// TwinCAT 3 PLC project Plc
// ProgramVersion: 3.1.4024.0
// libraries:
//   Tc2_Standard, * (Beckhoff Automation GmbH)
//   Tc2_System, * (Beckhoff Automation GmbH)
//   Tc3_Module, * (Beckhoff Automation GmbH)
// project tree:
//   OOP/Elements/ I_PushButton.TcIO, I_Sensor.TcIO, NormallyOpenPushButton.TcPOU, NormallyClosePushButton.TcPOU, NormallyOpenSensor.TcPOU, NormallyCloseSensor.TcPOU
//   OOP/Module/ I_Motor.TcIO, MotorControl.TcPOU, SortingConveyor.TcPOU
//   OOP/ PRG_OOPApproach.TcPOU
//   / PlcTask.TcTTO
//   POUs/ MAIN.TcPOU, PRG_SortingConveyor_proceduralApproach.TcPOU

CONFIGURATION Plc
    RESOURCE PLC ON TwinCAT3
        TASK PlcTask(INTERVAL := T#10ms, PRIORITY := 20);
        PROGRAM MAIN WITH PlcTask : MAIN;
    END_RESOURCE
END_CONFIGURATION

// ---- OOP/Elements/I_PushButton.TcIO
INTERFACE I_PushButton

PROPERTY PUBLIC isPressed : BOOL
GET
END_GET
END_PROPERTY

PROPERTY PUBLIC isReleased : BOOL
GET
END_GET
END_PROPERTY

END_INTERFACE

// ---- OOP/Elements/I_Sensor.TcIO
INTERFACE I_Sensor

PROPERTY PUBLIC isActive : BOOL
GET
END_GET
END_PROPERTY

PROPERTY PUBLIC isInactive : BOOL
GET
END_GET
END_PROPERTY

END_INTERFACE

// ---- OOP/Module/I_Motor.TcIO
INTERFACE I_Motor

METHOD PUBLIC Start
VAR_INPUT
END_VAR
END_METHOD

METHOD PUBLIC stop : BOOL
VAR_INPUT
END_VAR
END_METHOD

END_INTERFACE

// ---- POUs/MAIN.TcPOU
PROGRAM MAIN
VAR

END_VAR


	PRG_SortingConveyor_proceduralApproach();
	PRG_OOPApproach();

END_PROGRAM

// ---- POUs/PRG_SortingConveyor_proceduralApproach.TcPOU
PROGRAM PRG_SortingConveyor_proceduralApproach
VAR
	stop AT%I* : BOOL;
	emergency AT%I* : BOOL;
	start AT%I* : BOOL;
	productDetectedSensor AT%I* : BOOL;
	conveyorFullSensor AT%I* : BOOL;
	motorContactor AT%Q* : BOOL;
	conveyorControl: BOOL;

	timeout: TOF;	
END_VAR

	
IF (NOT stop) OR (NOT emergency) THEN
	conveyorControl	:=	FALSE;
ELSIF start AND (stop) AND (emergency) THEN
	conveyorControl	:=	TRUE;
END_IF
	
timeout(IN:= conveyorControl AND productDetectedSensor, PT:= T#5S, Q=> , ET=> );

motorContactor	:=	conveyorControl AND timeout.Q AND (NOT conveyorFullSensor);

END_PROGRAM

// ---- OOP/PRG_OOPApproach.TcPOU
PROGRAM PRG_OOPApproach
VAR
	stop : NormallyClosePushButton;
	emergency : NormallyClosePushButton;
	stopNO : NormallyOpenPushButton;
	emergencyNO : NormallyOpenPushButton;
	start : NormallyOpenPushButton;
	productDetectedSensor : NormallyOpenSensor;
	conveyorFullSensor : NormallyOpenSensor;
	motorContactor : MotorControl;
	
	SortingConveyor: SortingConveyor (stop, emergency, start, productDetectedSensor, conveyorFullSensor, motorContactor);
	
//	conveyorControl: BOOL;
//	timeout: TOF;	
	
	
	useSpareSensor: BOOL;
END_VAR

	
IF NOT useSpareSensor THEN
	SortingConveyor (	
		stop:= stop, 
		emergency:= emergency, 
		start:= start, 
		productDetectedSensor:= productDetectedSensor, 
		conveyorFullSensor:= conveyorFullSensor, 
		motorContactor:= motorContactor	);
ELSE
	SortingConveyor (	
		stop:= stopNO, 
		emergency:= emergencyNO, 
		start:= start, 
		productDetectedSensor:= productDetectedSensor, 
		conveyorFullSensor:= conveyorFullSensor, 
		motorContactor:= motorContactor	);	
END_IF


//	IF (stop.isPressed) OR (emergency.isPressed) THEN
//		conveyorControl	:=	FALSE;
//	ELSIF start.isPressed AND (stop.isReleased) AND (emergency.isReleased) THEN
//		conveyorControl	:=	TRUE;
//	END_IF
		
//	timeout(IN:= conveyorControl AND productDetectedSensor.isActive, PT:= T#5S, Q=> , ET=> );

//	IF conveyorControl AND timeout.Q AND (conveyorFullSensor.isInactive) THEN
//		motorContactor.Start();	
//	ELSE
//		motorContactor.Stop();	
//	END_IF

END_PROGRAM

// ---- OOP/Elements/NormallyClosePushButton.TcPOU
FUNCTION_BLOCK NormallyClosePushButton IMPLEMENTS I_PushButton
VAR
	input AT%I* : BOOL;
END_VAR

PROPERTY PUBLIC isPressed : BOOL
GET
isPressed	:=	NOT input;
END_GET
END_PROPERTY

PROPERTY PUBLIC isReleased : BOOL
GET
isReleased	:=	input;
END_GET
END_PROPERTY

END_FUNCTION_BLOCK

// ---- OOP/Elements/NormallyOpenPushButton.TcPOU
FUNCTION_BLOCK NormallyOpenPushButton IMPLEMENTS I_PushButton
VAR
	input AT%I* : BOOL;
END_VAR

PROPERTY PUBLIC isPressed : BOOL
GET
isPressed	:=	input;
END_GET
END_PROPERTY

PROPERTY PUBLIC isReleased : BOOL
GET
isReleased	:=	NOT input;
END_GET
END_PROPERTY

END_FUNCTION_BLOCK

// ---- OOP/Elements/NormallyOpenSensor.TcPOU
FUNCTION_BLOCK NormallyOpenSensor IMPLEMENTS I_Sensor
VAR
	input AT%I* : BOOL;
END_VAR

PROPERTY PUBLIC isActive : BOOL
GET
isActive	:=	input;
END_GET
END_PROPERTY

PROPERTY PUBLIC isInactive : BOOL
GET
isInactive	:=	NOT input;
END_GET
END_PROPERTY

END_FUNCTION_BLOCK

// ---- OOP/Module/MotorControl.TcPOU
FUNCTION_BLOCK MotorControl IMPLEMENTS I_Motor
VAR
	OnOff AT%Q* : BOOL;
END_VAR

METHOD PUBLIC Start
VAR_INPUT
END_VAR
OnOff	:=	TRUE;
END_METHOD

METHOD PUBLIC stop : BOOL
VAR_INPUT
END_VAR
OnOff := FALSE;
END_METHOD

END_FUNCTION_BLOCK

// ---- OOP/Module/SortingConveyor.TcPOU
FUNCTION_BLOCK SortingConveyor
VAR_INPUT
	stop : I_PushButton;
	emergency : I_PushButton;
	start : I_PushButton;
	productDetectedSensor : I_Sensor;
	conveyorFullSensor : I_Sensor;
	motorContactor : I_Motor;
END_VAR
VAR_OUTPUT
END_VAR
VAR	
	conveyorControl: BOOL;
	timeout: TOF;		
	
END_VAR

		
	IF (stop.isPressed) OR (emergency.isPressed) THEN
		conveyorControl	:=	FALSE;
	ELSIF start.isPressed AND (stop.isReleased) AND (emergency.isReleased) THEN
		conveyorControl	:=	TRUE;
	END_IF
		
	timeout(IN:= conveyorControl AND productDetectedSensor.isActive, PT:= T#5S, Q=> , ET=> );

	IF conveyorControl AND timeout.Q AND (conveyorFullSensor.isInactive) THEN
		motorContactor.Start();	
	ELSE
		motorContactor.Stop();	
	END_IF

METHOD FB_init : BOOL
VAR_INPUT
	bInitRetains : BOOL; // if TRUE, the retain variables are initialized (warm start / cold start)
	bInCopyCode : BOOL;  // if TRUE, the instance afterwards gets moved into the copy code (online change)

	stop : I_PushButton;
	emergency : I_PushButton;
	start : I_PushButton;
	productDetectedSensor : I_Sensor;
	conveyorFullSensor : I_Sensor;
	motorContactor : I_Motor;
	
END_VAR

	THIS^.stop 						:=	stop 					; 
	THIS^.emergency 				:=  emergency 				;
	THIS^.start 					:=  start 					;
	THIS^.productDetectedSensor 	:=  productDetectedSensor 	;
	THIS^.conveyorFullSensor 		:=  conveyorFullSensor 		;
	THIS^.motorContactor 			:=  motorContactor 			;
END_METHOD

END_FUNCTION_BLOCK

// ---- OOP/Elements/NormallyCloseSensor.TcPOU
FUNCTION_BLOCK NormallyCloseSensor IMPLEMENTS I_Sensor
VAR
	input AT%I* : BOOL;
END_VAR

PROPERTY PUBLIC isActive : BOOL
GET
isActive	:=	NOT input;
END_GET
END_PROPERTY

PROPERTY PUBLIC isInactive : BOOL
GET
isInactive	:=	input;
END_GET
END_PROPERTY

END_FUNCTION_BLOCK
